Fanuc KAREL source: kf00049.KL

-- PROVISIONAL review KL for V770-1; original PC SHA256 457ecae27cd3e4c0f81124cf2124ad00e50b52ac5ec12f6237d2af983863abd3
-- Incomplete behavior may be omitted. Consult companion uncertainty JSON. Do not deploy.
PROGRAM KF00049
%NOLOCKGROUP
VAR
  I : INTEGER
  J : INTEGER
  X : REAL
  Y : REAL
  B : BOOLEAN
  C : BOOLEAN
  TXT : STRING[80]
  TXT2 : STRING[80]
  STATUS : INTEGER
-- UNRESOLVED_DECL AI type=002010
-- UNRESOLVED_DECL BI type=002010
-- UNRESOLVED_DECL P type=000102
-- UNRESOLVED_DECL JP type=000199
-- UNRESOLVED_DECL PF type=000101
-- UNRESOLVED_DECL V1 type=000013
-- UNRESOLVED_DECL V2 type=000013
BEGIN
  -- UNRESOLVED_PC offsets 5-16; opcodes 2E,23
  -- UNRESOLVED_PC offsets 21-43; opcodes 21,40,41,41,42
  -- UNRESOLVED_PC offsets 48-65; opcodes 2E,23,7A,43
  -- UNRESOLVED_PC offsets 70-81; opcodes 2E,23
  -- UNRESOLVED_PC offsets 91-95; opcodes 7F
END KF00049
